FUNCTION_BLOCK fbTowerLightCtrl
VAR_INPUT

	bAlarmOccur : BOOL;
	bMainOnOff : BOOL;
	bAutoPreparationStart : BOOL;
	bAutoPreparationCompleted : BOOL;
	bAutoOriginStart : BOOL;
	bAutoOriginCompleted : BOOL;
	bAutoStart : BOOL;
	bAutoProgress : BOOL;
	bAutoCycleStop: BOOL;
	bManualMode : BOOL;



END_VAR
VAR_OUTPUT
	bTowerLightRED : BOOL;
	bTowerLightYELLOW : BOOL;
	bTowerLightGREEN : BOOL;

END_VAR
VAR

	AlwaysOn : BOOL := TRUE;

	T1: TON;
	T2: TON;
END_VAR

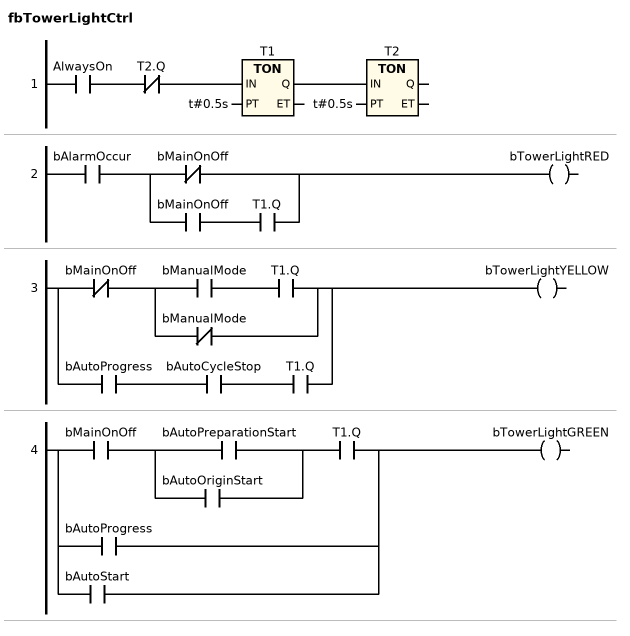
// NETWORK 1
T1(IN := AlwaysOn AND NOT T2.Q, PT := t#0.5s); // TON
T2(IN := T1.Q, PT := t#0.5s); // TON

// NETWORK 2
bTowerLightRED := bAlarmOccur AND (NOT bMainOnOff OR bMainOnOff AND T1.Q);

// NETWORK 3
bTowerLightYELLOW := NOT bMainOnOff AND (bManualMode AND T1.Q OR NOT bManualMode) OR bAutoProgress AND bAutoCycleStop AND T1.Q;

// NETWORK 4
bTowerLightGREEN := (bMainOnOff AND (bAutoPreparationStart OR bAutoOriginStart)) AND T1.Q OR bAutoProgress OR bAutoStart;

END_FUNCTION_BLOCK

(* stored: Version 1.1.0.1, ProductVersion 3.1.4024.12
   POU fbTowerLightCtrl: Id {7f5faa47-c722-40a4-ae06-0a188e35c347}, SpecialFunc None *)
